KUKA KRL program: SET_CP_STIFFNESS.src

&ACCESS RVO2
&REL 16
&PARAM TEMPLATE = C:\KRC\Roboter\Template\FunctionVorgabe
&PARAM EDITMASK = *
DEFFCT BOOL SET_CP_STIFFNESS(X_VAL:IN, Y_VAL:IN, Z_VAL:IN, A_VAL:IN, B_VAL:IN, C_VAL:IN )

REAL X_VAL, Y_VAL, Z_VAL
REAL A_VAL, B_VAL, C_VAL

$STIFFNESS.CPSTIFFNESS.X = X_VAL
$STIFFNESS.CPSTIFFNESS.Y = Y_VAL
$STIFFNESS.CPSTIFFNESS.Z = Z_VAL
$STIFFNESS.CPSTIFFNESS.A = A_VAL
$STIFFNESS.CPSTIFFNESS.B = B_VAL
$STIFFNESS.CPSTIFFNESS.C = C_VAL

$STIFFNESS.COMMIT = TRUE

RETURN TRUE

ENDFCT
